// Mitsubishi GX Works2 project: 闪烁控制   PLC: FX1S

PROGRAM MAIN
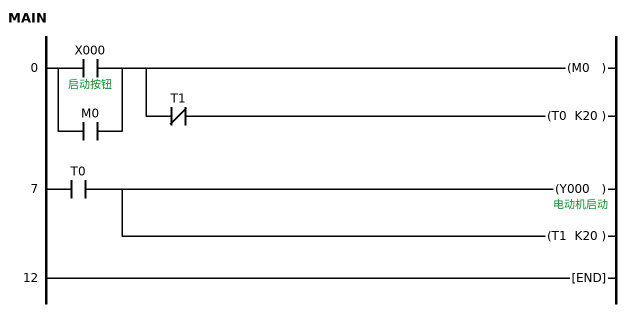
0     LD      X000  ; 启动按钮
      OR      M0
      OUT     M0
      ANI     T1
      OUT     T0 K20
7     LD      T0
      OUT     Y000  ; 电动机启动
      OUT     T1 K20
12    END
END_PROGRAM
